(* Logix 5000 project; controller DUNEW2PLC1 vendor 1 type 14 code 221 rev 33.11; software revision 33.00; part 3 of 7 *)
(* tags used below, declared in another part *)
   AbortActive : BOOL;
   CheckCurSeg : BOOL;
   CheckNextSeg : BOOL;
   CmdA_Accel : REAL;
   CmdA_CircleType : DINT;
   CmdA_Decel : REAL;
   CmdA_Direction : DINT;
   CmdA_JerkAccel : REAL;
   CmdA_JerkDecel : REAL;
   CmdA_SegType : DINT;
   CmdA_Speed : REAL;
   CmdA_TermType : SINT;
   CmdA_ViaCenter : REAL[2];
   CmdA_XY : REAL[2];
   CmdB_Accel : REAL;
   CmdB_CircleType : DINT;
   CmdB_Decel : REAL;
   CmdB_Direction : DINT;
   CmdB_JerkAccel : REAL;
   CmdB_JerkDecel : REAL;
   CmdB_SegType : DINT;
   CmdB_Speed : REAL;
   CmdB_TermType : SINT;
   CmdB_ViaCenter : REAL[2];
   CmdB_XY : REAL[2];
   CmdTolerance : DINT;
   CurSeg : MotionSeg;
   DoneONS_A : BOOL;
   DoneONS_B : BOOL;
   EnqueueReq : BOOL;
   FaultCode : DINT;
   FlipToA : BOOL;
   FlipToB : BOOL;
   IssueCurPulse : BOOL;
   IssueNextPulse : BOOL;
   LoadCurReq : BOOL;
   LoadNextReq : BOOL;
   MoveA : MOTION_INSTRUCTION;
   MoveB : MOTION_INSTRUCTION;
   NextSeg : MotionSeg;
   PrepCurMove : BOOL;
   PrepNextMove : BOOL;
   QueueCtl : CONTROL;
   QueueEmpty : BOOL;
   RotateMoves : BOOL;
   RotateONS_AtoB : BOOL;
   RotateONS_BtoA : BOOL;
   StartNextA_ONS : BOOL;
   StartNextB_ONS : BOOL;
   UseAasCurrent : BOOL;
   WaitCurAxisOn : BOOL;
   WaitNextAxisOn : BOOL;
   x_axis_mso : MOTION_INSTRUCTION;
   y_axis_mso : MOTION_INSTRUCTION;
   AbortQueue : BOOL;
   ActiveSeq : DINT;
   APA_IS_VERTICAL : BOOL;
   CurIssueAckTON : TIMER;
   CurIssued : BOOL;
   ERROR_CODE : DINT;
   IncomingSegReqID : DINT;
   LastIncomingSegReqID : DINT;
   NextIssueAckTON : TIMER;
   NextIssued : BOOL;
   NEXTSTATE : DINT;
   PendingSeq : DINT;
   QueueDiag_AbortActive : BOOL;
   QueueDiag_ActiveSeq : DINT;
   QueueDiag_CheckCurSeg : BOOL;
   QueueDiag_CheckNextSeg : BOOL;
   QueueDiag_CmdA_SegType : DINT;
   QueueDiag_CmdB_SegType : DINT;
   QueueDiag_CurSeg_SegType : DINT;
   QueueDiag_CurSeg_Seq : DINT;
   QueueDiag_CurSeg_Speed : DINT;
   QueueDiag_CurSeg_TermType : DINT;
   QueueDiag_CurSeg_Valid : BOOL;
   QueueDiag_CurSeg_X : DINT;
   QueueDiag_CurSeg_Y : DINT;
   QueueDiag_FaultCode : DINT;
   QueueDiag_FlipToA : BOOL;
   QueueDiag_FlipToB : BOOL;
   QueueDiag_IssueCurPulse : BOOL;
   QueueDiag_IssueNextPulse : BOOL;
   QueueDiag_LoadCurReq : BOOL;
   QueueDiag_LoadNextReq : BOOL;
   QueueDiag_MoveA_DN : BOOL;
   QueueDiag_MoveA_ER : BOOL;
   QueueDiag_MoveA_ERRID : DINT;
   QueueDiag_MoveA_EXERR : DINT;
   QueueDiag_MoveA_IP : BOOL;
   QueueDiag_MoveA_PC : BOOL;
   QueueDiag_MoveB_DN : BOOL;
   QueueDiag_MoveB_ER : BOOL;
   QueueDiag_MoveB_ERRID : DINT;
   QueueDiag_MoveB_EXERR : DINT;
   QueueDiag_MoveB_IP : BOOL;
   QueueDiag_MoveB_PC : BOOL;
   QueueDiag_NextSeg_SegType : DINT;
   QueueDiag_NextSeg_Seq : DINT;
   QueueDiag_NextSeg_Speed : DINT;
   QueueDiag_NextSeg_TermType : DINT;
   QueueDiag_NextSeg_Valid : BOOL;
   QueueDiag_NextSeg_X : DINT;
   QueueDiag_NextSeg_Y : DINT;
   QueueDiag_PendingSeq : DINT;
   QueueDiag_PrepCurMove : BOOL;
   QueueDiag_PrepNextMove : BOOL;
   QueueDiag_QueueCtl_DN : BOOL;
   QueueDiag_QueueCtl_EM : BOOL;
   QueueDiag_QueueCtl_EN : BOOL;
   QueueDiag_QueueCtl_ER : BOOL;
   QueueDiag_QueueCtl_EU : BOOL;
   QueueDiag_QueueCtl_IN : BOOL;
   QueueDiag_QueueCtl_LEN : DINT;
   QueueDiag_QueueCtl_POS : DINT;
   QueueDiag_QueueCtl_UL : BOOL;
   QueueDiag_RotateMoves : BOOL;
   QueueDiag_UseAasCurrent : BOOL;
   QueueDiag_WaitCurAxisOn : BOOL;
   QueueDiag_WaitNextAxisOn : BOOL;
   QueueFault : BOOL;
   QueueStopRequest : BOOL;
   SegQueue : MotionSeg[32];
   StartQueuedPath : BOOL;
   X_axis : AXIS_CIP_DRIVE;
   X_Y : COORDINATE_SYSTEM;
   Y_axis : AXIS_CIP_DRIVE;
(* queued_motion, continued *)

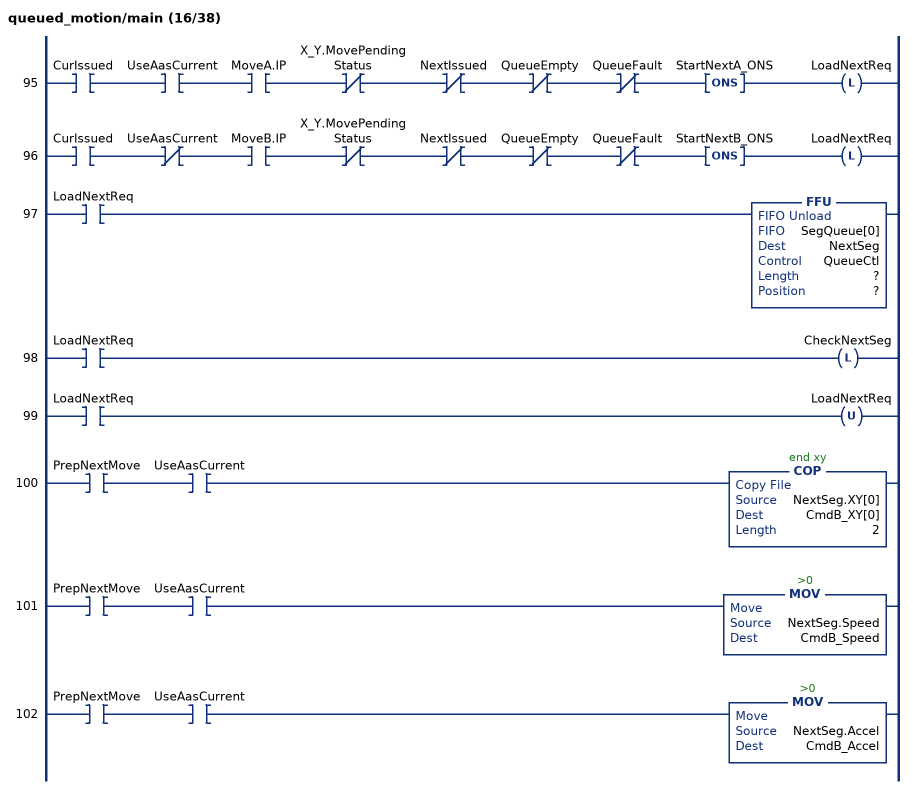
   [picture p44: queued_motion/main rungs 95-102]
   95: XIC(CurIssued)XIC(UseAasCurrent)XIC(MoveA.IP)XIO(X_Y.MovePendingStatus)XIO(NextIssued)XIO(QueueEmpty)XIO(QueueFault)ONS(StartNextA_ONS)OTL(LoadNextReq);
   96: XIC(CurIssued)XIO(UseAasCurrent)XIC(MoveB.IP)XIO(X_Y.MovePendingStatus)XIO(NextIssued)XIO(QueueEmpty)XIO(QueueFault)ONS(StartNextB_ONS)OTL(LoadNextReq);
   97: XIC(LoadNextReq)FFU(SegQueue[0],NextSeg,QueueCtl,?,?);
   98: XIC(LoadNextReq)OTL(CheckNextSeg);
   99: XIC(LoadNextReq)OTU(LoadNextReq);
   100: XIC(PrepNextMove)XIC(UseAasCurrent)COP(NextSeg.XY[0],CmdB_XY[0],2);
   101: XIC(PrepNextMove)XIC(UseAasCurrent)MOV(NextSeg.Speed,CmdB_Speed);
   102: XIC(PrepNextMove)XIC(UseAasCurrent)MOV(NextSeg.Accel,CmdB_Accel);
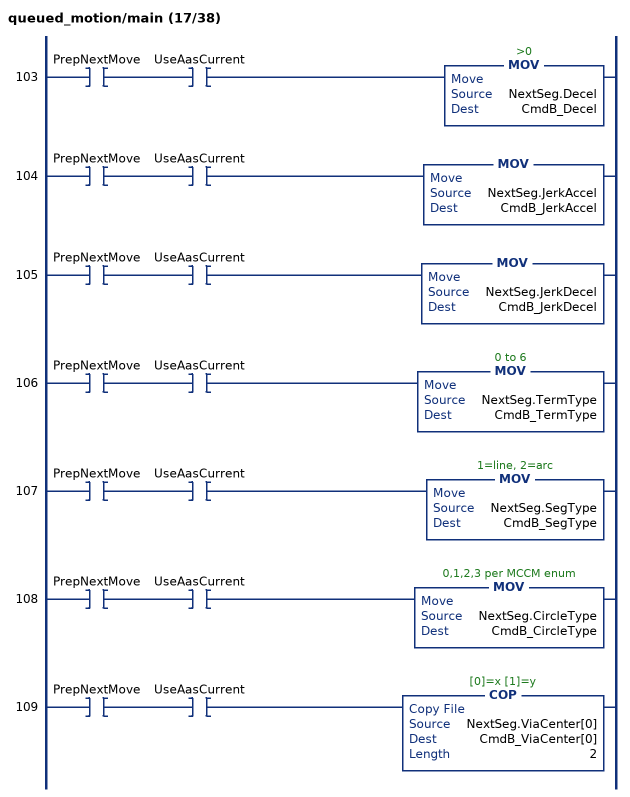
   103: XIC(PrepNextMove)XIC(UseAasCurrent)MOV(NextSeg.Decel,CmdB_Decel);
   104: XIC(PrepNextMove)XIC(UseAasCurrent)MOV(NextSeg.JerkAccel,CmdB_JerkAccel);
   105: XIC(PrepNextMove)XIC(UseAasCurrent)MOV(NextSeg.JerkDecel,CmdB_JerkDecel);
   106: XIC(PrepNextMove)XIC(UseAasCurrent)MOV(NextSeg.TermType,CmdB_TermType);
   107: XIC(PrepNextMove)XIC(UseAasCurrent)MOV(NextSeg.SegType,CmdB_SegType);
   108: XIC(PrepNextMove)XIC(UseAasCurrent)MOV(NextSeg.CircleType,CmdB_CircleType);
   109: XIC(PrepNextMove)XIC(UseAasCurrent)COP(NextSeg.ViaCenter[0],CmdB_ViaCenter[0],2);
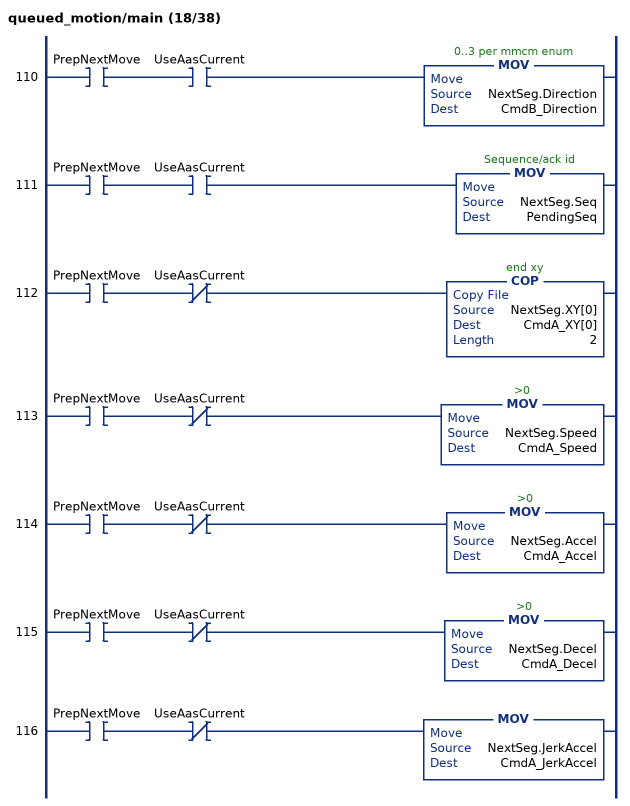
   110: XIC(PrepNextMove)XIC(UseAasCurrent)MOV(NextSeg.Direction,CmdB_Direction);
   111: XIC(PrepNextMove)XIC(UseAasCurrent)MOV(NextSeg.Seq,PendingSeq);
   112: XIC(PrepNextMove)XIO(UseAasCurrent)COP(NextSeg.XY[0],CmdA_XY[0],2);
   113: XIC(PrepNextMove)XIO(UseAasCurrent)MOV(NextSeg.Speed,CmdA_Speed);
   114: XIC(PrepNextMove)XIO(UseAasCurrent)MOV(NextSeg.Accel,CmdA_Accel);
   115: XIC(PrepNextMove)XIO(UseAasCurrent)MOV(NextSeg.Decel,CmdA_Decel);
   116: XIC(PrepNextMove)XIO(UseAasCurrent)MOV(NextSeg.JerkAccel,CmdA_JerkAccel);
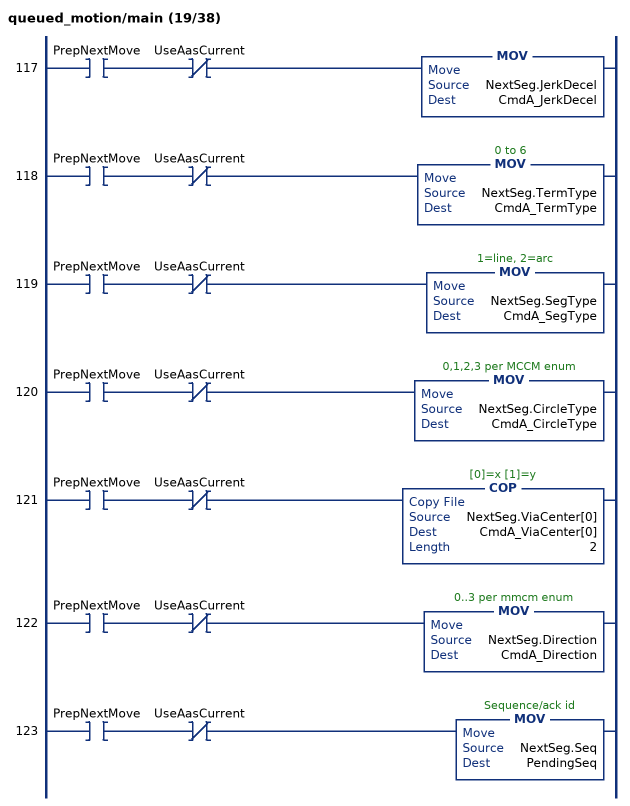
   117: XIC(PrepNextMove)XIO(UseAasCurrent)MOV(NextSeg.JerkDecel,CmdA_JerkDecel);
   118: XIC(PrepNextMove)XIO(UseAasCurrent)MOV(NextSeg.TermType,CmdA_TermType);
   119: XIC(PrepNextMove)XIO(UseAasCurrent)MOV(NextSeg.SegType,CmdA_SegType);
   120: XIC(PrepNextMove)XIO(UseAasCurrent)MOV(NextSeg.CircleType,CmdA_CircleType);
   121: XIC(PrepNextMove)XIO(UseAasCurrent)COP(NextSeg.ViaCenter[0],CmdA_ViaCenter[0],2);
   122: XIC(PrepNextMove)XIO(UseAasCurrent)MOV(NextSeg.Direction,CmdA_Direction);
   123: XIC(PrepNextMove)XIO(UseAasCurrent)MOV(NextSeg.Seq,PendingSeq);
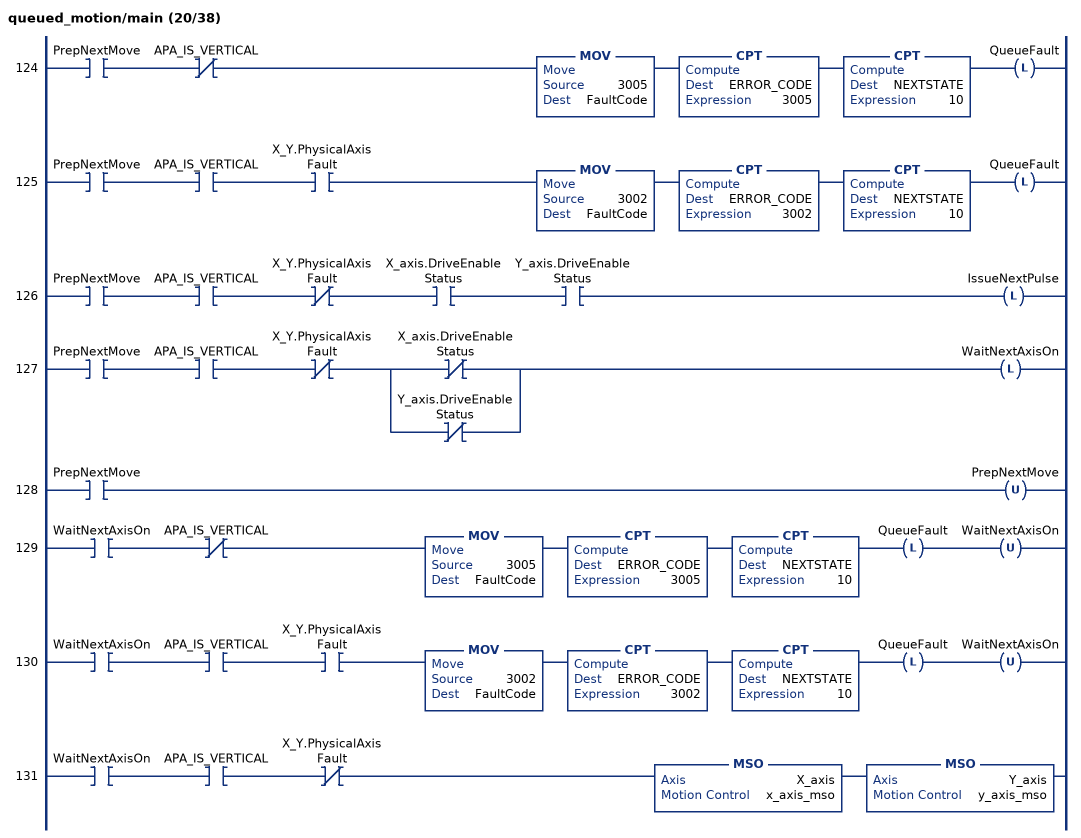
   124: XIC(PrepNextMove)XIO(APA_IS_VERTICAL)MOV(3005,FaultCode)CPT(ERROR_CODE,3005)CPT(NEXTSTATE,10)OTL(QueueFault);
   125: XIC(PrepNextMove)XIC(APA_IS_VERTICAL)XIC(X_Y.PhysicalAxisFault)MOV(3002,FaultCode)CPT(ERROR_CODE,3002)CPT(NEXTSTATE,10)OTL(QueueFault);
   126: XIC(PrepNextMove)XIC(APA_IS_VERTICAL)XIO(X_Y.PhysicalAxisFault)XIC(X_axis.DriveEnableStatus)XIC(Y_axis.DriveEnableStatus)OTL(IssueNextPulse);
   127: XIC(PrepNextMove)XIC(APA_IS_VERTICAL)XIO(X_Y.PhysicalAxisFault)[XIO(X_axis.DriveEnableStatus) ,XIO(Y_axis.DriveEnableStatus) ]OTL(WaitNextAxisOn);
   128: XIC(PrepNextMove)OTU(PrepNextMove);
   129: XIC(WaitNextAxisOn)XIO(APA_IS_VERTICAL)MOV(3005,FaultCode)CPT(ERROR_CODE,3005)CPT(NEXTSTATE,10)OTL(QueueFault)OTU(WaitNextAxisOn);
   130: XIC(WaitNextAxisOn)XIC(APA_IS_VERTICAL)XIC(X_Y.PhysicalAxisFault)MOV(3002,FaultCode)CPT(ERROR_CODE,3002)CPT(NEXTSTATE,10)OTL(QueueFault)OTU(WaitNextAxisOn);
   131: XIC(WaitNextAxisOn)XIC(APA_IS_VERTICAL)XIO(X_Y.PhysicalAxisFault)MSO(X_axis,x_axis_mso)MSO(Y_axis,y_axis_mso);
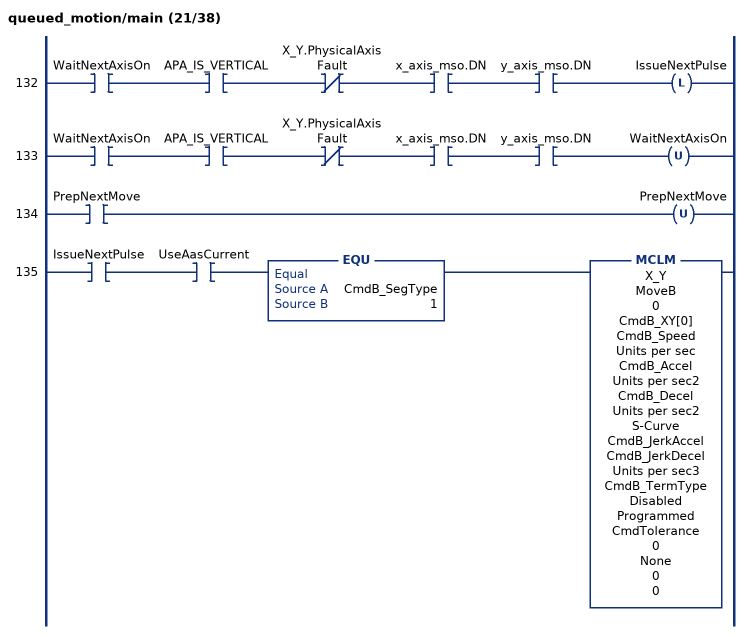
   132: XIC(WaitNextAxisOn)XIC(APA_IS_VERTICAL)XIO(X_Y.PhysicalAxisFault)XIC(x_axis_mso.DN)XIC(y_axis_mso.DN)OTL(IssueNextPulse);
   133: XIC(WaitNextAxisOn)XIC(APA_IS_VERTICAL)XIO(X_Y.PhysicalAxisFault)XIC(x_axis_mso.DN)XIC(y_axis_mso.DN)OTU(WaitNextAxisOn);
   134: XIC(PrepNextMove)OTU(PrepNextMove);
   135: XIC(IssueNextPulse)XIC(UseAasCurrent)EQU(CmdB_SegType,1)MCLM(X_Y,MoveB,0,CmdB_XY[0],CmdB_Speed,Units per sec,CmdB_Accel,Units per sec2,CmdB_Decel,Units per sec2,S-Curve,CmdB_JerkAccel,CmdB_JerkDecel,Units per sec3,CmdB_TermType,Disabled,Programmed,CmdTolerance,0,None,0,0);
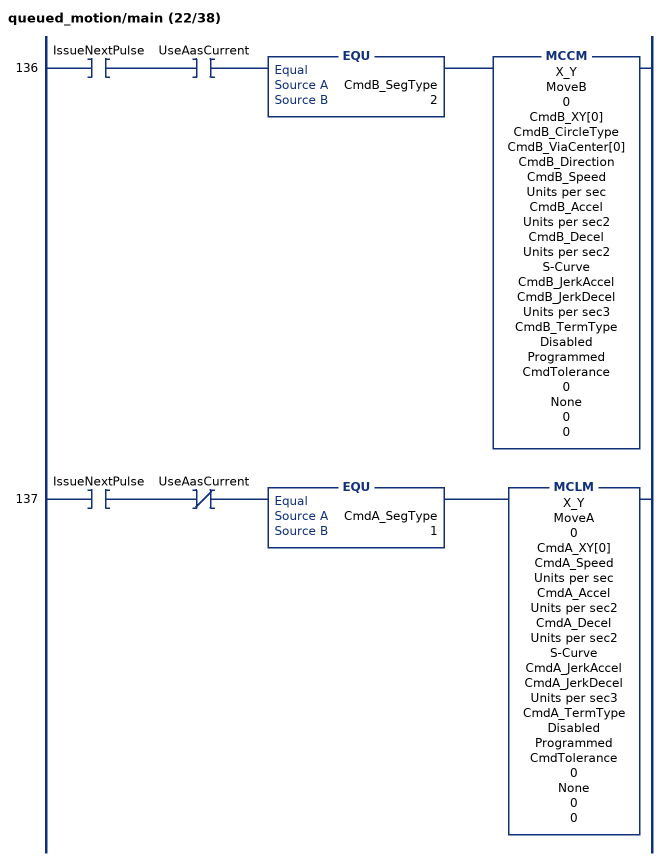
   136: XIC(IssueNextPulse)XIC(UseAasCurrent)EQU(CmdB_SegType,2)MCCM(X_Y,MoveB,0,CmdB_XY[0],CmdB_CircleType,CmdB_ViaCenter[0],CmdB_Direction,CmdB_Speed,Units per sec,CmdB_Accel,Units per sec2,CmdB_Decel,Units per sec2,S-Curve,CmdB_JerkAccel,CmdB_JerkDecel,Units per sec3,CmdB_TermType,Disabled,Programmed,CmdTolerance,0,None,0,0);
   137: XIC(IssueNextPulse)XIO(UseAasCurrent)EQU(CmdA_SegType,1)MCLM(X_Y,MoveA,0,CmdA_XY[0],CmdA_Speed,Units per sec,CmdA_Accel,Units per sec2,CmdA_Decel,Units per sec2,S-Curve,CmdA_JerkAccel,CmdA_JerkDecel,Units per sec3,CmdA_TermType,Disabled,Programmed,CmdTolerance,0,None,0,0);
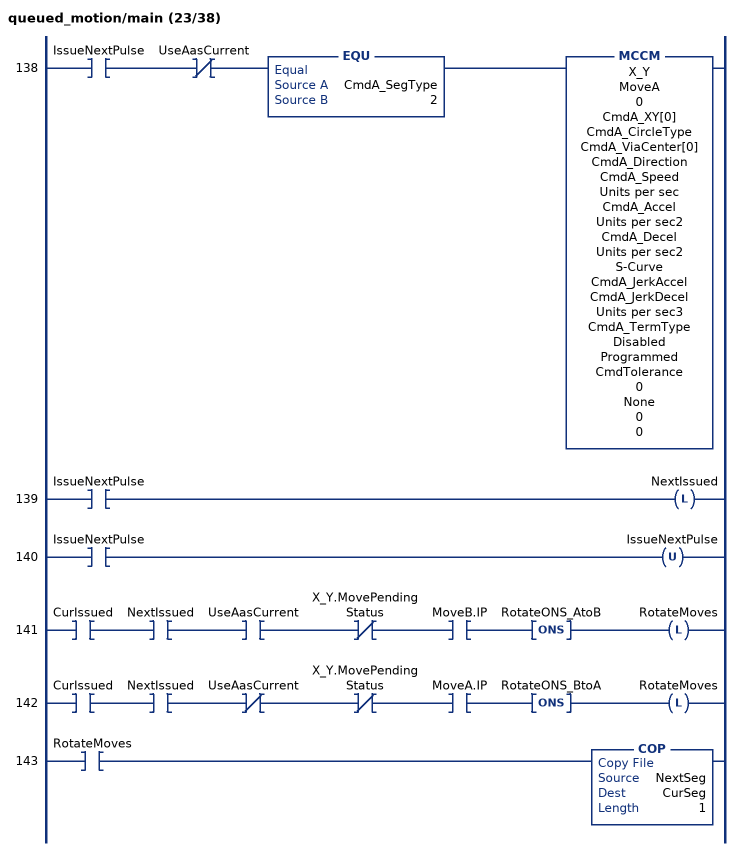
   138: XIC(IssueNextPulse)XIO(UseAasCurrent)EQU(CmdA_SegType,2)MCCM(X_Y,MoveA,0,CmdA_XY[0],CmdA_CircleType,CmdA_ViaCenter[0],CmdA_Direction,CmdA_Speed,Units per sec,CmdA_Accel,Units per sec2,CmdA_Decel,Units per sec2,S-Curve,CmdA_JerkAccel,CmdA_JerkDecel,Units per sec3,CmdA_TermType,Disabled,Programmed,CmdTolerance,0,None,0,0);
   139: XIC(IssueNextPulse)OTL(NextIssued);
   140: XIC(IssueNextPulse)OTU(IssueNextPulse);
   141: XIC(CurIssued)XIC(NextIssued)XIC(UseAasCurrent)XIO(X_Y.MovePendingStatus)XIC(MoveB.IP)ONS(RotateONS_AtoB)OTL(RotateMoves);
   142: XIC(CurIssued)XIC(NextIssued)XIO(UseAasCurrent)XIO(X_Y.MovePendingStatus)XIC(MoveA.IP)ONS(RotateONS_BtoA)OTL(RotateMoves);
   143: XIC(RotateMoves)COP(NextSeg,CurSeg,1);
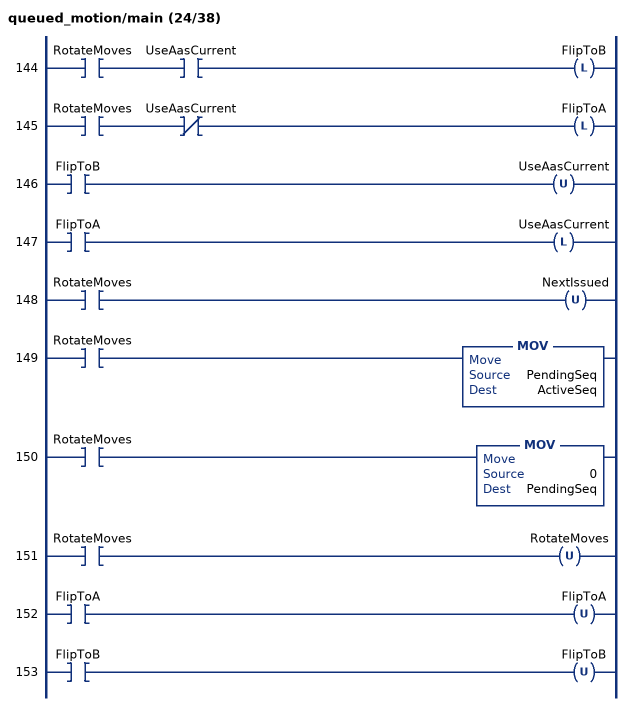
   144: XIC(RotateMoves)XIC(UseAasCurrent)OTL(FlipToB);
   145: XIC(RotateMoves)XIO(UseAasCurrent)OTL(FlipToA);
   146: XIC(FlipToB)OTU(UseAasCurrent);
   147: XIC(FlipToA)OTL(UseAasCurrent);
   148: XIC(RotateMoves)OTU(NextIssued);
   149: XIC(RotateMoves)MOV(PendingSeq,ActiveSeq);
   150: XIC(RotateMoves)MOV(0,PendingSeq);
   151: XIC(RotateMoves)OTU(RotateMoves);
   152: XIC(FlipToA)OTU(FlipToA);
   153: XIC(FlipToB)OTU(FlipToB);
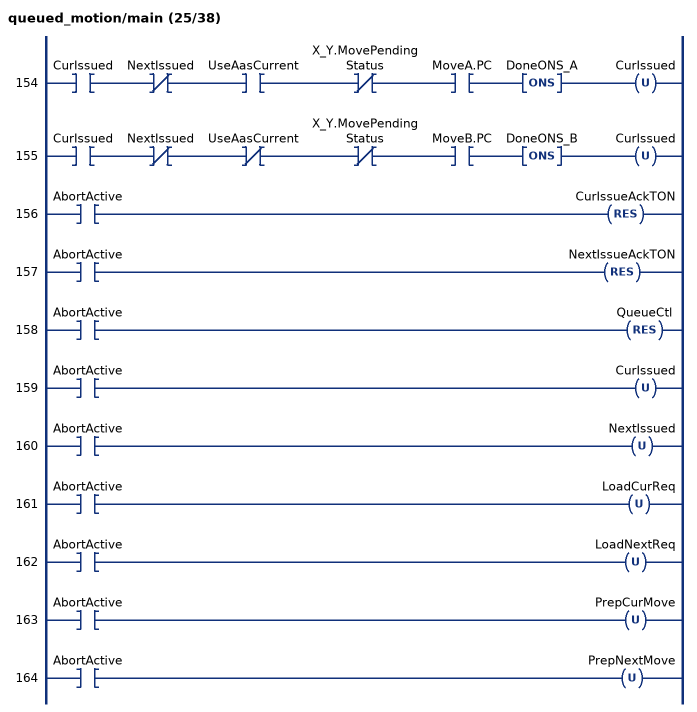
   154: XIC(CurIssued)XIO(NextIssued)XIC(UseAasCurrent)XIO(X_Y.MovePendingStatus)XIC(MoveA.PC)ONS(DoneONS_A)OTU(CurIssued);
   155: XIC(CurIssued)XIO(NextIssued)XIO(UseAasCurrent)XIO(X_Y.MovePendingStatus)XIC(MoveB.PC)ONS(DoneONS_B)OTU(CurIssued);
   156: XIC(AbortActive)RES(CurIssueAckTON);
   157: XIC(AbortActive)RES(NextIssueAckTON);
   158: XIC(AbortActive)RES(QueueCtl);
   159: XIC(AbortActive)OTU(CurIssued);
   160: XIC(AbortActive)OTU(NextIssued);
   161: XIC(AbortActive)OTU(LoadCurReq);
   162: XIC(AbortActive)OTU(LoadNextReq);
   163: XIC(AbortActive)OTU(PrepCurMove);
   164: XIC(AbortActive)OTU(PrepNextMove);
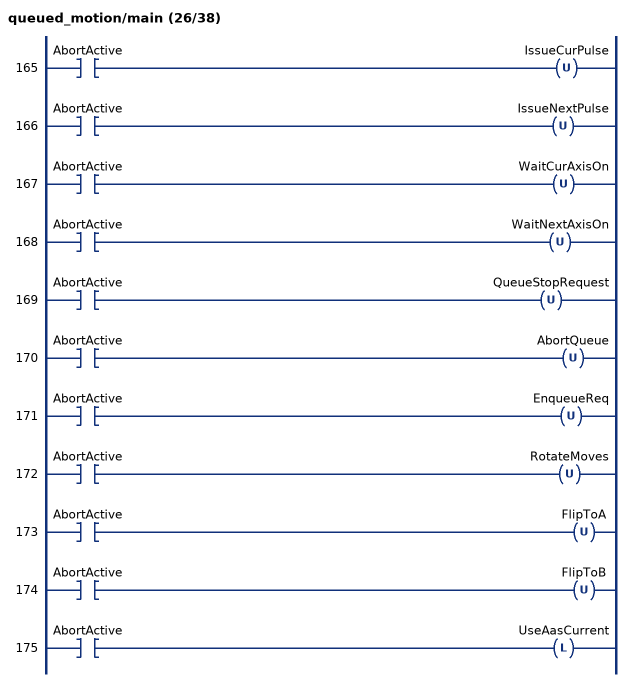
   165: XIC(AbortActive)OTU(IssueCurPulse);
   166: XIC(AbortActive)OTU(IssueNextPulse);
   167: XIC(AbortActive)OTU(WaitCurAxisOn);
   168: XIC(AbortActive)OTU(WaitNextAxisOn);
   169: XIC(AbortActive)OTU(QueueStopRequest);
   170: XIC(AbortActive)OTU(AbortQueue);
   171: XIC(AbortActive)OTU(EnqueueReq);
   172: XIC(AbortActive)OTU(RotateMoves);
   173: XIC(AbortActive)OTU(FlipToA);
   174: XIC(AbortActive)OTU(FlipToB);
   175: XIC(AbortActive)OTL(UseAasCurrent);
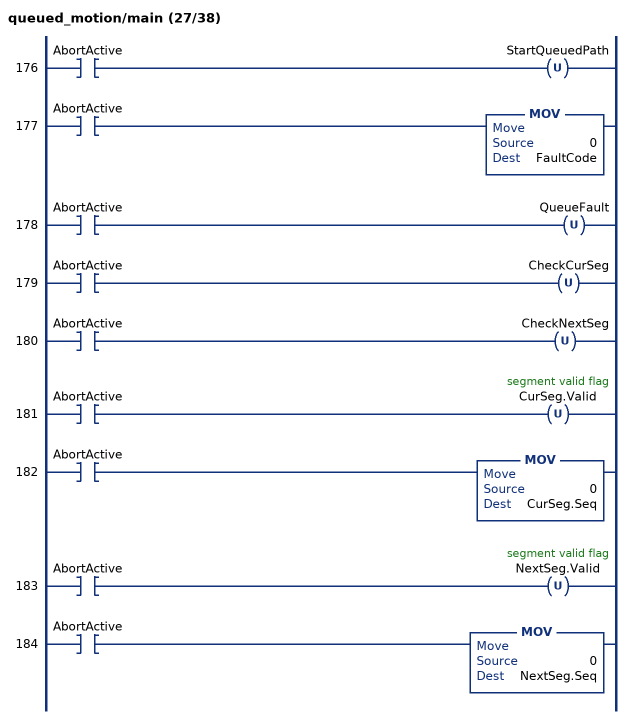
   176: XIC(AbortActive)OTU(StartQueuedPath);
   177: XIC(AbortActive)MOV(0,FaultCode);
   178: XIC(AbortActive)OTU(QueueFault);
   179: XIC(AbortActive)OTU(CheckCurSeg);
   180: XIC(AbortActive)OTU(CheckNextSeg);
   181: XIC(AbortActive)OTU(CurSeg.Valid);
   182: XIC(AbortActive)MOV(0,CurSeg.Seq);
   183: XIC(AbortActive)OTU(NextSeg.Valid);
   184: XIC(AbortActive)MOV(0,NextSeg.Seq);
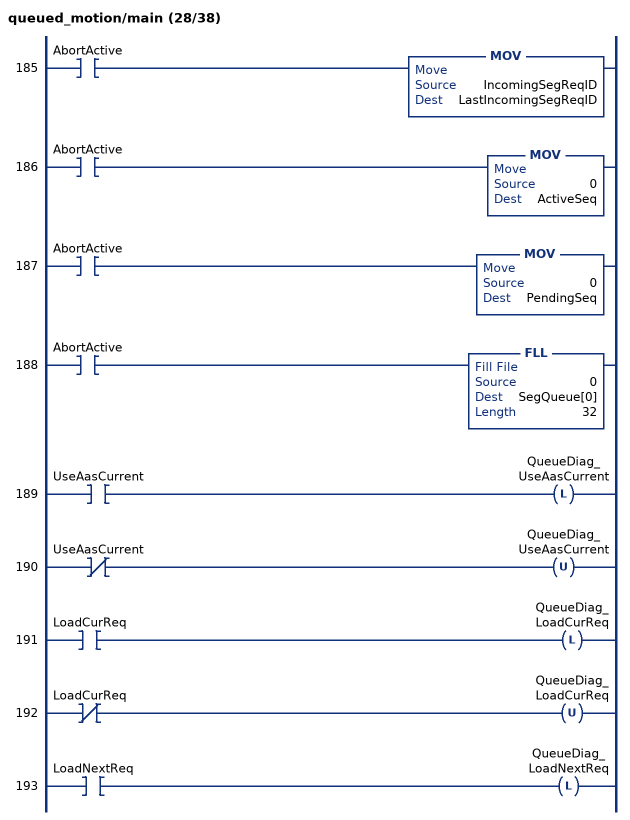
   185: XIC(AbortActive)MOV(IncomingSegReqID,LastIncomingSegReqID);
   186: XIC(AbortActive)MOV(0,ActiveSeq);
   187: XIC(AbortActive)MOV(0,PendingSeq);
   188: XIC(AbortActive)FLL(0,SegQueue[0],32);
   189: XIC(UseAasCurrent)OTL(QueueDiag_UseAasCurrent);
   190: XIO(UseAasCurrent)OTU(QueueDiag_UseAasCurrent);
   191: XIC(LoadCurReq)OTL(QueueDiag_LoadCurReq);
   192: XIO(LoadCurReq)OTU(QueueDiag_LoadCurReq);
   193: XIC(LoadNextReq)OTL(QueueDiag_LoadNextReq);
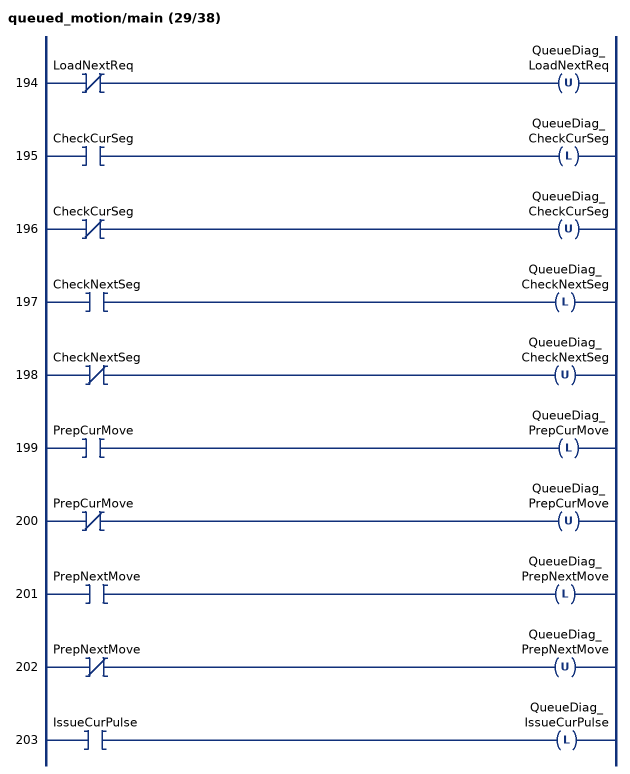
   194: XIO(LoadNextReq)OTU(QueueDiag_LoadNextReq);
   195: XIC(CheckCurSeg)OTL(QueueDiag_CheckCurSeg);
   196: XIO(CheckCurSeg)OTU(QueueDiag_CheckCurSeg);
   197: XIC(CheckNextSeg)OTL(QueueDiag_CheckNextSeg);
   198: XIO(CheckNextSeg)OTU(QueueDiag_CheckNextSeg);
   199: XIC(PrepCurMove)OTL(QueueDiag_PrepCurMove);
   200: XIO(PrepCurMove)OTU(QueueDiag_PrepCurMove);
   201: XIC(PrepNextMove)OTL(QueueDiag_PrepNextMove);
   202: XIO(PrepNextMove)OTU(QueueDiag_PrepNextMove);
   203: XIC(IssueCurPulse)OTL(QueueDiag_IssueCurPulse);
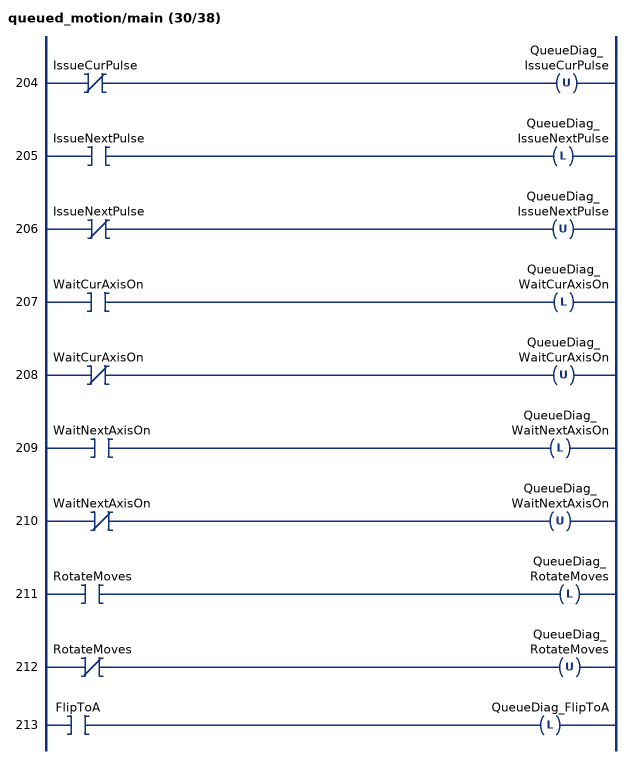
   204: XIO(IssueCurPulse)OTU(QueueDiag_IssueCurPulse);
   205: XIC(IssueNextPulse)OTL(QueueDiag_IssueNextPulse);
   206: XIO(IssueNextPulse)OTU(QueueDiag_IssueNextPulse);
   207: XIC(WaitCurAxisOn)OTL(QueueDiag_WaitCurAxisOn);
   208: XIO(WaitCurAxisOn)OTU(QueueDiag_WaitCurAxisOn);
   209: XIC(WaitNextAxisOn)OTL(QueueDiag_WaitNextAxisOn);
   210: XIO(WaitNextAxisOn)OTU(QueueDiag_WaitNextAxisOn);
   211: XIC(RotateMoves)OTL(QueueDiag_RotateMoves);
   212: XIO(RotateMoves)OTU(QueueDiag_RotateMoves);
   213: XIC(FlipToA)OTL(QueueDiag_FlipToA);
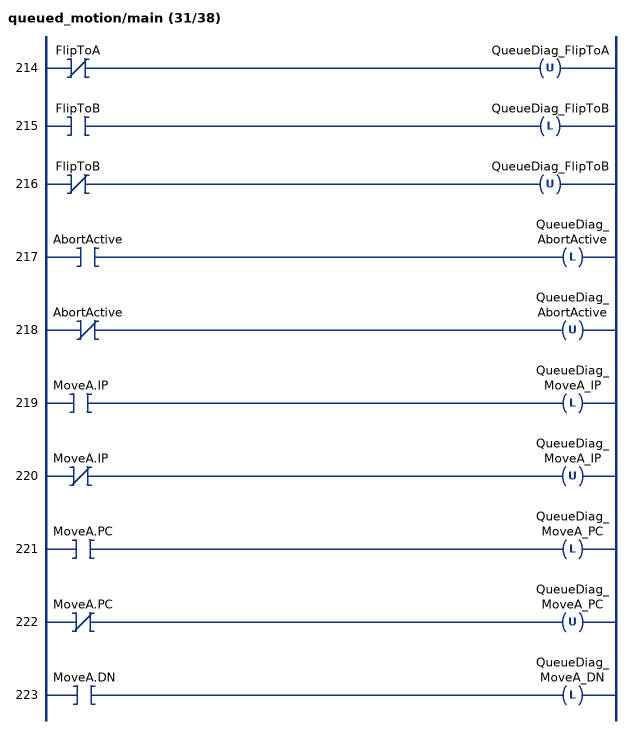
   214: XIO(FlipToA)OTU(QueueDiag_FlipToA);
   215: XIC(FlipToB)OTL(QueueDiag_FlipToB);
   216: XIO(FlipToB)OTU(QueueDiag_FlipToB);
   217: XIC(AbortActive)OTL(QueueDiag_AbortActive);
   218: XIO(AbortActive)OTU(QueueDiag_AbortActive);
   219: XIC(MoveA.IP)OTL(QueueDiag_MoveA_IP);
   220: XIO(MoveA.IP)OTU(QueueDiag_MoveA_IP);
   221: XIC(MoveA.PC)OTL(QueueDiag_MoveA_PC);
   222: XIO(MoveA.PC)OTU(QueueDiag_MoveA_PC);
   223: XIC(MoveA.DN)OTL(QueueDiag_MoveA_DN);
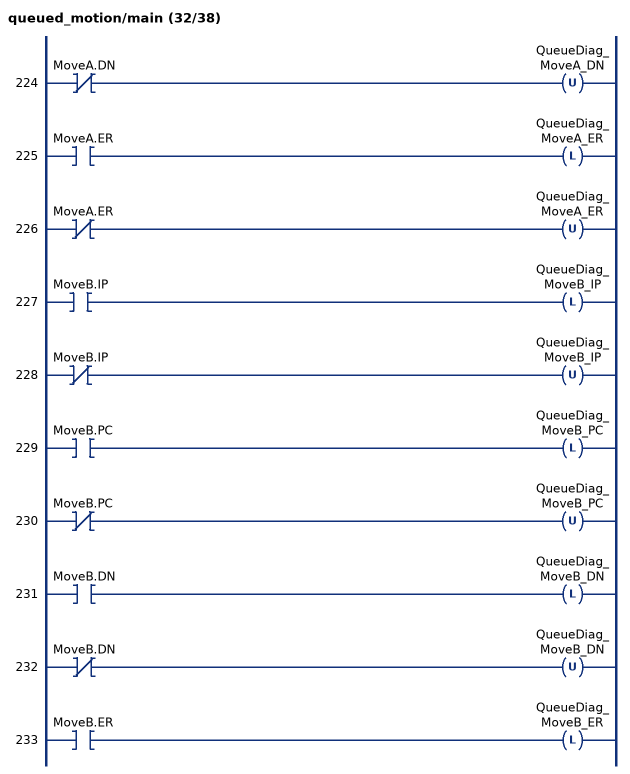
   224: XIO(MoveA.DN)OTU(QueueDiag_MoveA_DN);
   225: XIC(MoveA.ER)OTL(QueueDiag_MoveA_ER);
   226: XIO(MoveA.ER)OTU(QueueDiag_MoveA_ER);
   227: XIC(MoveB.IP)OTL(QueueDiag_MoveB_IP);
   228: XIO(MoveB.IP)OTU(QueueDiag_MoveB_IP);
   229: XIC(MoveB.PC)OTL(QueueDiag_MoveB_PC);
   230: XIO(MoveB.PC)OTU(QueueDiag_MoveB_PC);
   231: XIC(MoveB.DN)OTL(QueueDiag_MoveB_DN);
   232: XIO(MoveB.DN)OTU(QueueDiag_MoveB_DN);
   233: XIC(MoveB.ER)OTL(QueueDiag_MoveB_ER);
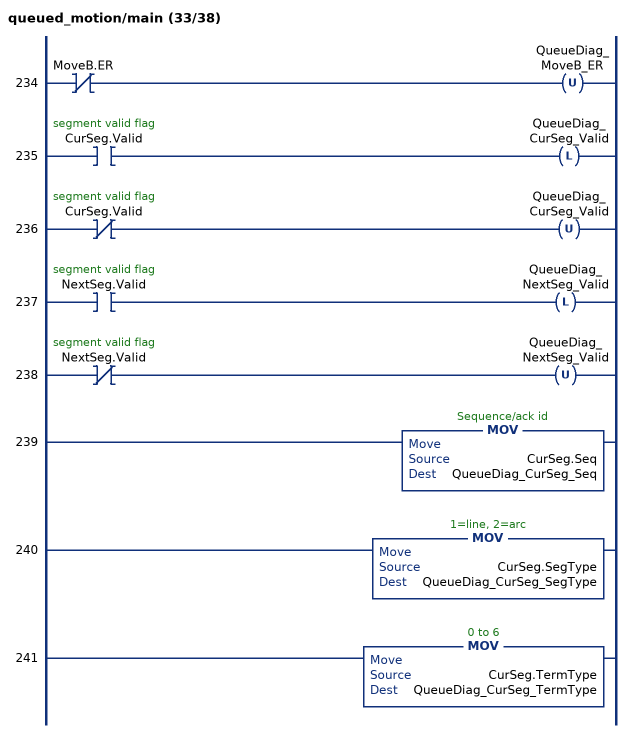
   234: XIO(MoveB.ER)OTU(QueueDiag_MoveB_ER);
   235: XIC(CurSeg.Valid)OTL(QueueDiag_CurSeg_Valid);
   236: XIO(CurSeg.Valid)OTU(QueueDiag_CurSeg_Valid);
   237: XIC(NextSeg.Valid)OTL(QueueDiag_NextSeg_Valid);
   238: XIO(NextSeg.Valid)OTU(QueueDiag_NextSeg_Valid);
   239: MOV(CurSeg.Seq,QueueDiag_CurSeg_Seq);
   240: MOV(CurSeg.SegType,QueueDiag_CurSeg_SegType);
   241: MOV(CurSeg.TermType,QueueDiag_CurSeg_TermType);
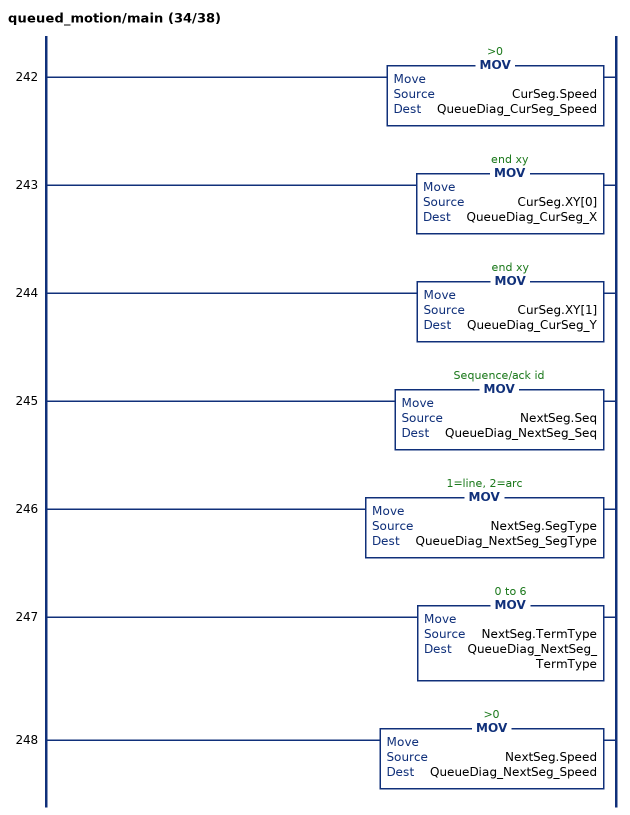
   242: MOV(CurSeg.Speed,QueueDiag_CurSeg_Speed);
   243: MOV(CurSeg.XY[0],QueueDiag_CurSeg_X);
   244: MOV(CurSeg.XY[1],QueueDiag_CurSeg_Y);
   245: MOV(NextSeg.Seq,QueueDiag_NextSeg_Seq);
   246: MOV(NextSeg.SegType,QueueDiag_NextSeg_SegType);
   247: MOV(NextSeg.TermType,QueueDiag_NextSeg_TermType);
   248: MOV(NextSeg.Speed,QueueDiag_NextSeg_Speed);
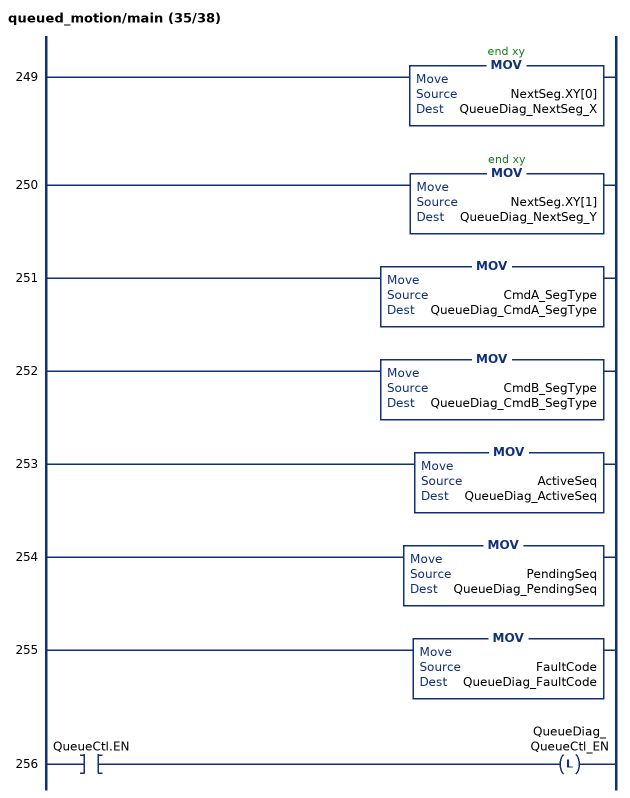
   249: MOV(NextSeg.XY[0],QueueDiag_NextSeg_X);
   250: MOV(NextSeg.XY[1],QueueDiag_NextSeg_Y);
   251: MOV(CmdA_SegType,QueueDiag_CmdA_SegType);
   252: MOV(CmdB_SegType,QueueDiag_CmdB_SegType);
   253: MOV(ActiveSeq,QueueDiag_ActiveSeq);
   254: MOV(PendingSeq,QueueDiag_PendingSeq);
   255: MOV(FaultCode,QueueDiag_FaultCode);
   256: XIC(QueueCtl.EN)OTL(QueueDiag_QueueCtl_EN);
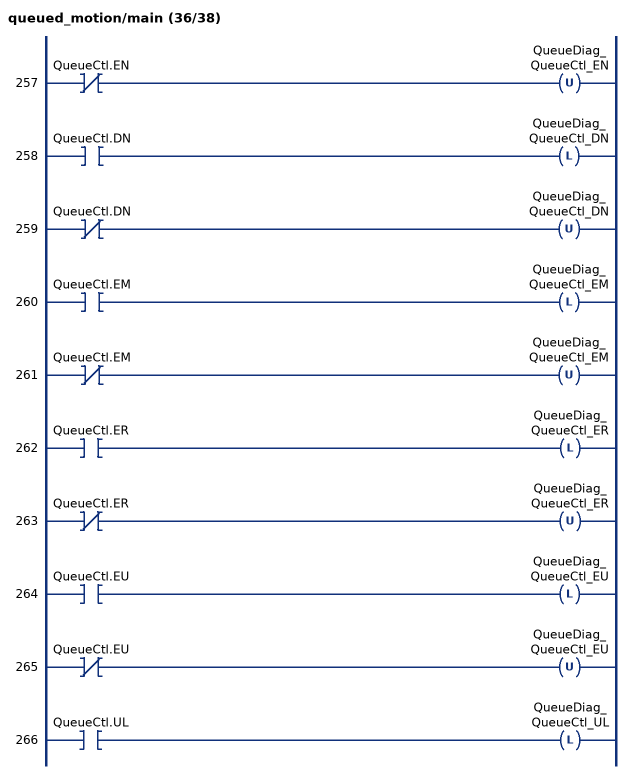
   257: XIO(QueueCtl.EN)OTU(QueueDiag_QueueCtl_EN);
   258: XIC(QueueCtl.DN)OTL(QueueDiag_QueueCtl_DN);
   259: XIO(QueueCtl.DN)OTU(QueueDiag_QueueCtl_DN);
   260: XIC(QueueCtl.EM)OTL(QueueDiag_QueueCtl_EM);
   261: XIO(QueueCtl.EM)OTU(QueueDiag_QueueCtl_EM);
   262: XIC(QueueCtl.ER)OTL(QueueDiag_QueueCtl_ER);
   263: XIO(QueueCtl.ER)OTU(QueueDiag_QueueCtl_ER);
   264: XIC(QueueCtl.EU)OTL(QueueDiag_QueueCtl_EU);
   265: XIO(QueueCtl.EU)OTU(QueueDiag_QueueCtl_EU);
   266: XIC(QueueCtl.UL)OTL(QueueDiag_QueueCtl_UL);
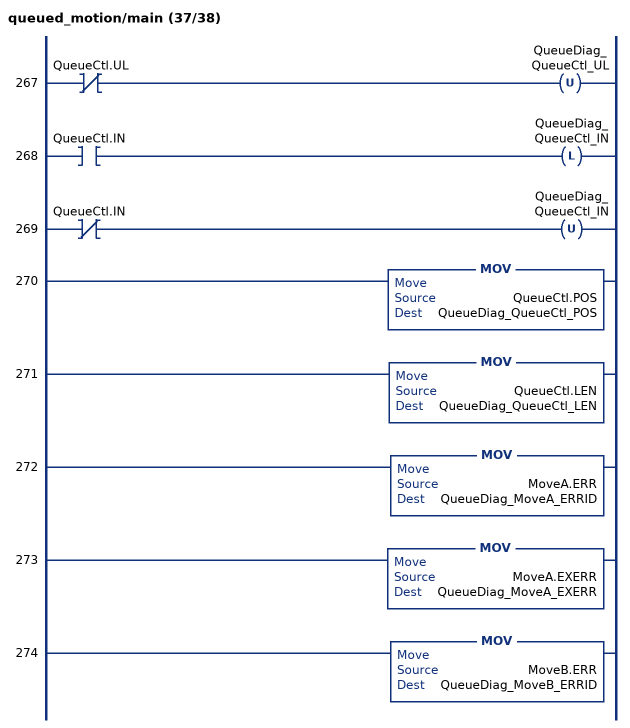
   267: XIO(QueueCtl.UL)OTU(QueueDiag_QueueCtl_UL);
   268: XIC(QueueCtl.IN)OTL(QueueDiag_QueueCtl_IN);
   269: XIO(QueueCtl.IN)OTU(QueueDiag_QueueCtl_IN);
   270: MOV(QueueCtl.POS,QueueDiag_QueueCtl_POS);
   271: MOV(QueueCtl.LEN,QueueDiag_QueueCtl_LEN);
   272: MOV(MoveA.ERR,QueueDiag_MoveA_ERRID);
   273: MOV(MoveA.EXERR,QueueDiag_MoveA_EXERR);
   274: MOV(MoveB.ERR,QueueDiag_MoveB_ERRID);
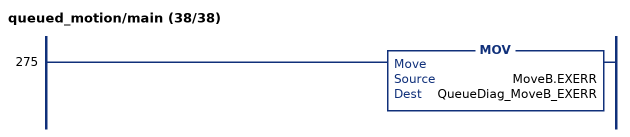
   275: MOV(MoveB.EXERR,QueueDiag_MoveB_EXERR);
END_ROUTINE
